Yaskawa INFORM job: DEMO_NAIHAN_0625_2PAINT_2.JBI

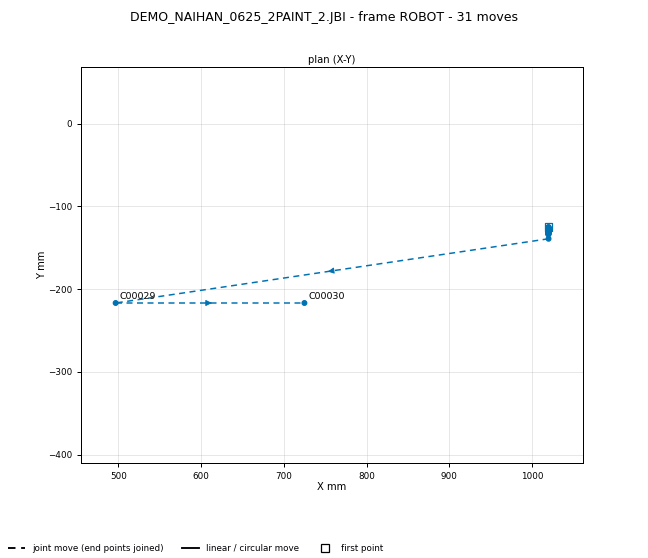
[picture p0: tool path of DEMO_NAIHAN_0625_2PAINT_2.JBI in frame ROBOT, 31 of 31 moves have a stored position in this frame; points joined in program order, loops and branches not executed]
/JOB
//NAME DEMO_NAIHAN_0625_2PAINT2
//POS
///NPOS 31,0,0,0,0,0
///TOOL 1
///USER 0
///POSTYPE ROBOT
///RECTAN
///RCONF 1,0,0,0,1,0,0,0,0,0,0,0,0,0,0,0,0,0,0,0,0,0,0,0
C00000=1019.977,-124.933,387.526,-23.937,21.717,-44.638
C00001=1019.973,-125.261,387.548,-23.936,21.717,-44.643
C00002=1019.970,-125.590,387.569,-23.936,21.719,-44.647
C00003=1019.967,-125.917,387.591,-23.935,21.719,-44.652
C00004=1019.963,-126.246,387.613,-23.935,21.720,-44.657
C00005=1019.959,-126.574,387.635,-23.934,21.720,-44.662
C00006=1019.956,-126.902,387.657,-23.933,21.720,-44.667
C00007=1019.952,-127.230,387.679,-23.933,21.721,-44.671
C00008=1019.949,-127.558,387.701,-23.932,21.721,-44.676
C00009=1019.945,-127.885,387.722,-23.931,21.722,-44.680
C00010=1019.941,-128.214,387.743,-23.931,21.723,-44.686
C00011=1019.937,-128.542,387.766,-23.930,21.723,-44.689
C00012=1019.934,-128.870,387.787,-23.929,21.723,-44.695
C00013=1019.930,-129.198,387.809,-23.929,21.725,-44.699
C00014=1019.926,-129.526,387.831,-23.928,21.724,-44.704
C00015=1019.923,-129.854,387.853,-23.928,21.726,-44.708
C00016=1019.919,-130.182,387.875,-23.927,21.726,-44.713
C00017=1019.915,-130.510,387.897,-23.927,21.726,-44.717
C00018=1019.912,-130.838,387.917,-23.926,21.727,-44.723
C00019=1019.908,-131.166,387.939,-23.926,21.728,-44.726
C00020=1019.903,-131.494,387.961,-23.925,21.728,-44.732
C00021=1019.900,-131.822,387.983,-23.924,21.729,-44.736
C00022=1019.896,-132.150,388.005,-23.924,21.729,-44.741
C00023=1019.892,-132.478,388.026,-23.923,21.730,-44.745
C00024=1019.889,-132.806,388.048,-23.922,21.731,-44.750
C00025=1019.884,-133.133,388.069,-23.922,21.731,-44.754
C00026=1019.880,-133.462,388.092,-23.921,21.731,-44.759
C00027=1019.877,-133.790,388.112,-23.921,21.732,-44.763
C00028=1020.037,-139.035,388.427,-23.921,21.732,-44.763
///USER 0
///POSTYPE ROBOT
///RECTAN
///RCONF 1,0,0,0,0,0,0,0,0,0,0,0,0,0,0,0,0,0,0,0,0,0,0,0
C00029=496.664,-216.680,394.500,-180.000,-0.000,-0.000
C00030=724.889,-216.680,394.500,-180.000,-0.000,-0.000
//INST
///DATE 2021/06/25 14:57
///ATTR SC,RW,RJ
////FRAME ROBOT
///GROUP1 RB1
NOP
MOVL C00000 V=800.0 PL=0
MOVL C00001 V=800.0 PL=0
MOVL C00002 V=800.0 PL=0
MOVL C00003 V=800.0 PL=0
MOVL C00004 V=800.0 PL=0
MOVL C00005 V=800.0 PL=0
MOVL C00006 V=800.0 PL=0
MOVL C00007 V=800.0 PL=0
MOVL C00008 V=800.0 PL=0
MOVL C00009 V=800.0 PL=0
MOVL C00010 V=800.0 PL=0
MOVL C00011 V=800.0 PL=0
MOVL C00012 V=800.0 PL=0
MOVL C00013 V=800.0 PL=0
MOVL C00014 V=800.0 PL=0
MOVL C00015 V=800.0 PL=0
MOVL C00016 V=800.0 PL=0
MOVL C00017 V=800.0 PL=0
MOVL C00018 V=800.0 PL=0
MOVL C00019 V=800.0 PL=0
MOVL C00020 V=800.0 PL=0
MOVL C00021 V=800.0 PL=0
MOVL C00022 V=800.0 PL=0
MOVL C00023 V=800.0 PL=0
MOVL C00024 V=800.0 PL=0
MOVL C00025 V=800.0 PL=0
MOVL C00026 V=800.0 PL=0
MOVL C00027 V=800.0 PL=0
'CALL JOB: TOOL OFF
MOVJ C00028 VJ=25.00 PL=0
'Path End
MOVJ C00029 VJ=100.00 PL=0
MOVJ C00030 VJ=100.00 PL=0
END
